(*
SPDX-FileCopyrightText: © 2026 Oleksandr Tiutyk <trofimich@gmail.com>
SPDX-License-Identifier: MIT
License: https://opensource.org/license/mit
*)

TYPE HMI_INTERSECTION_CONTROLLER_COMMANDS :
STRUCT
	TurnOn : BOOL;
	TurnOff : BOOL;

	SetYellowFlashingModeOn : BOOL;
	SetYellowFlashingModeOff : BOOL;
	
	SetSwitchingSpeedCorrectionPercent : BOOL;
	SwitchingSpeedCorrectionPercent : SPEED_CORRECTION_PERCENT;
	
	ThrowExceptionInDemoExceptionGenerator : BOOL;
	ExceptionMessage : STRING(255) := 'Test error message';
	ExceptionIsCritical : BOOL;
END_STRUCT
END_TYPE

(* stored: Version 1.1.0.1
   DUT HMI_INTERSECTION_CONTROLLER_COMMANDS: Id {d2a31d68-a228-45de-800d-93de748e46ae} *)
